FUNCTION Prepare_Date_Time : STRING(255)
VAR_INPUT
	plcDT									: ARRAY[0..6] OF DINT;
	
END_VAR
VAR
	str_DT									: Tc2_Utilities.TIMESTRUCT;
	tmp_str									: STRING(255);
	tmp_result								: STRING(255);
END_VAR

//fb_Time();
	str_DT.wYear			:=DINT_TO_WORD(plcDT[0]);
	str_DT.wMonth			:=DINT_TO_WORD(plcDT[1]);
	str_DT.wDay				:=DINT_TO_WORD(plcDT[2]);
	str_DT.wHour			:=DINT_TO_WORD(plcDT[3]);
	str_DT.wMinute			:=DINT_TO_WORD(plcDT[4]);
	str_DT.wSecond			:=DINT_TO_WORD(plcDT[5]);
	str_DT.wMilliseconds	:=DINT_TO_WORD(plcDT[6]);
	
	
	tmp_result := Tc2_Standard.CONCAT('DATE ', WORD_TO_STRING(str_DT.wYear MOD 100));
	tmp_result := Tc2_Standard.CONCAT(tmp_result, '-');
	tmp_str    := WORD_TO_STRING(str_DT.wMonth);
	IF Tc2_Standard.LEN(tmp_str) < 2 THEN
		tmp_str := Tc2_Standard.CONCAT('0', tmp_str);
	END_IF;
	tmp_result := Tc2_Standard.CONCAT(tmp_result, tmp_str);
	
	tmp_result := Tc2_Standard.CONCAT(tmp_result, '-');
	tmp_str    := WORD_TO_STRING(str_DT.wDay);
	IF Tc2_Standard.LEN(tmp_str) < 2 THEN
		tmp_str := Tc2_Standard.CONCAT('0', tmp_str);
	END_IF;
	tmp_result := Tc2_Standard.CONCAT(tmp_result, tmp_str);

	tmp_result := Tc2_Standard.CONCAT(tmp_result, '  TIME ');
	tmp_str    := WORD_TO_STRING(str_DT.wHour);
	IF Tc2_Standard.LEN(tmp_str) < 2 THEN
		tmp_str := Tc2_Standard.CONCAT('0', tmp_str);
	END_IF;
	tmp_result := Tc2_Standard.CONCAT(tmp_result, tmp_str);

	tmp_result := Tc2_Standard.CONCAT(tmp_result, ':');
	tmp_str    := WORD_TO_STRING(str_DT.wMinute);
	IF Tc2_Standard.LEN(tmp_str) < 2 THEN
		tmp_str := Tc2_Standard.CONCAT('0', tmp_str);
	END_IF;
	tmp_result := Tc2_Standard.CONCAT(tmp_result, tmp_str);

	tmp_result := Tc2_Standard.CONCAT(tmp_result, ':');
	tmp_str    := WORD_TO_STRING(str_DT.wSecond);
	IF Tc2_Standard.LEN(tmp_str) < 2 THEN
		tmp_str := Tc2_Standard.CONCAT('0', tmp_str);
	END_IF;
	tmp_result := Tc2_Standard.CONCAT(tmp_result, tmp_str);
	
	tmp_result := Tc2_Standard.CONCAT(tmp_result, ':');
	tmp_str    := WORD_TO_STRING(str_DT.wMilliseconds);
	IF Tc2_Standard.LEN(tmp_str) = 1 THEN
		tmp_str := Tc2_Standard.CONCAT('00', tmp_str);
	END_IF;
	IF Tc2_Standard.LEN(tmp_str) = 2 THEN
		tmp_str := Tc2_Standard.CONCAT('0', tmp_str);
	END_IF;
	tmp_result := Tc2_Standard.CONCAT(tmp_result, tmp_str);	
	Prepare_Date_Time := tmp_result;

END_FUNCTION

(* stored: Version 1.1.0.1, ProductVersion 3.1.4024.12
   POU Prepare_Date_Time: Id {a05ba712-ab28-4751-afe3-5501d19dd475}, SpecialFunc None *)
